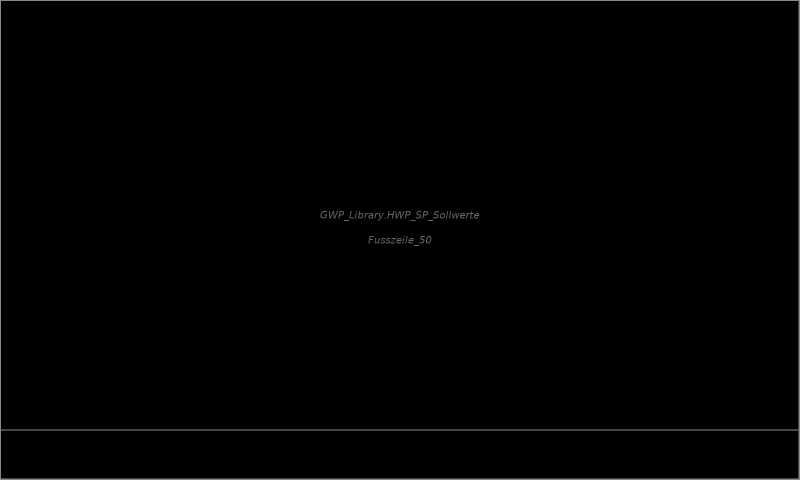
VISUALIZATION HWP_SP_Sollwerte  // 800x480
    Frame (0,0 800x430)
        shows GWP_Library.HWP_SP_Sollwerte(FB_HWP_SP := Main.HWP_SP_0, FB_Kreis_3KO := Main.Kreis_3KO_0)
    Frame (0,0 800x480)
        shows Fusszeile_50()
END_VISUALIZATION

(* stored: Version 1.1.0.1, ProductVersion 3.1.4022.6
   Visu HWP_SP_Sollwerte: Id {50df6d79-a110-447b-ae9b-5fc5fef08f70} *)
